(* PLC project io_on_off_pump, Dassault Systèmes ControlBuild 2024x *)
(* stored: creationDateTime 2023-10-03T11:12:48-01:00 *)

PROGRAM panel
  VAR_OUTPUT
    onPB : BOOL := false;
    offPB : BOOL := false;
  END_VAR

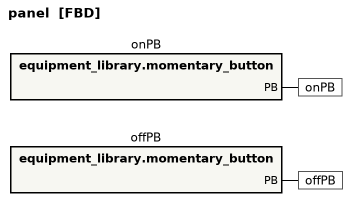
(* FBD diagram, written out as Structured Text *)
onPB();
onPB := onPB.PB;
offPB();
offPB := offPB.PB;
END_PROGRAM

(* Integrated object C/C+OP of an on/off pump *)
PROGRAM io_library.io_on_off_pump
  VAR_INPUT
    acknowledgePB : BOOL := false;
  END_VAR
  VAR_INPUT
    autoMode : BOOL := false;
    manualMode : BOOL := false;
  END_VAR
  VAR_INPUT
    autoCmd : BOOL := false;
  END_VAR
  VAR_INPUT
    inputFlow : REAL := 0.0;
  END_VAR
  VAR_OUTPUT
    generalFault : BOOL := false;
    speedVal : REAL := 0.0;
    outputFlow : REAL := 0.0;
  END_VAR

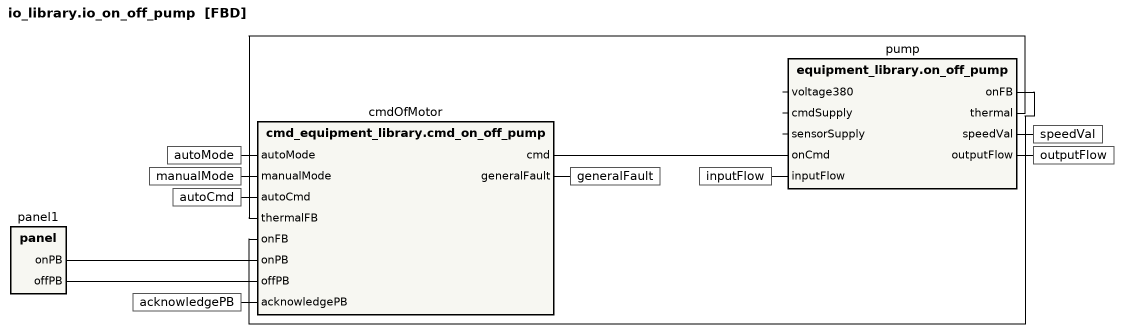
(* FBD diagram, written out as Structured Text *)
pump(onCmd := cmdOfMotor.cmd, inputFlow := inputFlow);
panel1();
cmdOfMotor(autoMode := autoMode, manualMode := manualMode, autoCmd := autoCmd, thermalFB := pump.thermal, onFB := pump.onFB, onPB := panel1.onPB, offPB := panel1.offPB, acknowledgePB := acknowledgePB);
generalFault := cmdOfMotor.generalFault;
speedVal := pump.speedVal;
outputFlow := pump.outputFlow;
END_PROGRAM
